// SIMATIC S7-200 project (STEP 7-Micro/WIN), CPU 224 REL 01.10

ORGANIZATION_BLOCK MAIN:OB1
TITLE=我使用这个PLC程序控制一台自动化纺织机，用于在纺织厂的织造车间。
// 系统支持多种运行模式，通过控制模式VB801选择运行模式，VB801的值必须在1到4之间。
// 程序通过高速计数器HC1记录织造的纬纱数量，计数器C10记录纬纱切换次数，用于监控生产进度和切换情况。
// 程序涉及的物理设备包括纺织机、电机、纬纱检测传感器、经纱检测传感器、启动按钮、停止按钮、纬纱切换执行器和PLC控制器。
// 系统支持多种运行模式，操作员通过控制模式选择器选择模式，其值必须在1到4之间。
// 织造通过启动按钮触发，当经纱检测传感器确认经纱正常时，运行标志置位以开始织造过程。操作员按下停止按钮时，系统复位运行标志以停止织造。纬纱切换由纬纱切换执行器控制，只有在纬纱检测传感器检测到纬纱到位时才会触发，确保切换动作准确无误。纬纱切换执行器在织造过程中由系统根据运行状态自动激活，以支持纬纱的连续切换。纬纱检测传感器用于监测纬纱的到位情况，触发计时器以协调织造节奏。系统通过经纱检测传感器监控经纱状态，若异常触发经停位标志，调用经停位子程序暂停织造。
// 为满足手动调试需求，系统支持点动控制，通过点动起输出和点动停输出实现，分别调用点动起子程序和点动停子程序，在点动模式下独立触发。若纬纱出现故障，故障标志置位，系统进入纬停状态，调用纬停位子程序安全停车并等待处理。
// 
// 
BEGIN
Network 1 // NETWORK TITLE (single line)
LD     SM0.1
CALL   初始化:SBR0
MOVB   0, MB0
?000
Network 2
LD     SM0.0
MOVB   VB93, VB153
Network 3
LDN    V142.2
MOVW   VW244, VW144
Network 4
LD     V142.2
EU
MOVW   VW144, VW244
MOVD   16#1000, VD14
R      V142.2, 1
Network 5
LDB<=  VB801, 1
=      M18.1
MOVB   1, VB801
Network 6
LDB=   VB801, 2
=      M18.2
Network 7
LDB=   VB801, 3
=      M18.3
Network 8
LDB>=  VB801, 4
=      M18.4
MOVB   4, VB801
Network 9
LD     I0.4
ED
O      M12.0
AN     T6
=      M12.0
Network 10
LD     T6
R      T6, 1
Network 11
LD     M12.0
TONR   T6, +900
Network 12
LD     I1.5
AN     M12.0
EU
CALL   启动:SBR3
Network 13
LD     I1.5
ED
CALL   即停位:SBR8
MOVD   16#20000000, VD14
Network 14
LDB=   VB811, 1
JMP    1
Network 15
LDB<>  VB811, 1
DISI
Network 16
LD     M0.0
MOVD   16#40000000, VD14
R      M0.0, 1
Network 17
// vw44 vw144 当前纬纱序号 VW244同色纬纱根数 
LD     M22.0
MOVD   16#4000000, VD14
MOVW   VW44, VW144
MOVD   &VB1000, AC3
+I     VW84, AC3
MOVB   *AC3, VB253
MOVW   +0, VW244
R      M22.0, 1
Network 18
LD     SM0.0
MOVW   VW5118, VW5116
-I     +1, VW5116
Network 19
LD     M0.1
MOVD   16#8000000, VD14
R      M0.1, 1
Network 20
LD     V228.2
MOVD   16#20000000, VD14
R      V228.2, 1
Network 21
LDB<=  VB201, 1
=      M20.1
MOVB   1, VB201
Network 22
LDB=   VB201, 2
=      M20.2
Network 23
LDB=   VB201, 3
=      M20.3
Network 24
LDB=   VB201, 4
=      M20.4
Network 25
LDB=   VB201, 5
=      M20.5
Network 26
LDB>=  VB201, 3
=      M20.3
MOVB   3, VB201
Network 27
LD     M20.1
EU
S      C10, 1
MOVW   +1, C2
MOVB   16#0, VB1101
MOVB   16#1, VB1103
Network 28
LD     M20.2
EU
S      C10, 1
S      C12, 1
MOVW   +1, C10
MOVW   +1, C12
MOVB   16#1, VB1101
MOVB   16#1, VB1103
Network 29
LD     M20.3
EU
S      C10, 1
S      C12, 1
MOVW   +2, C10
MOVW   +2, C12
MOVB   16#2, VB1101
MOVB   16#2, VB1103
Network 30
LDB=   VB231, 1
S      M18.7, 1
Network 31
LDB=   VB231, 0
R      M18.7, 1
Network 32
LD     M18.7
MOVW   VW220, VW4468
*I     +10, VW4468
Network 33
LDN    M18.7
ITD    VW220, AC0
DTR    AC0, VD1196
MOVR   VD1196, VD1192
*R     39.37, VD1192
ROUND  VD1192, VD4466
Network 34
LD     M0.2
MOVD   16#10000000, VD14
R      M0.2, 1
Network 35
LD     V160.2
MOVD   16#20000000, VD14
R      V160.2, 1
Network 36
LD     SM0.0
MOVW   VW162, VW5102
-I     +102, VW5102
MOVW   VW182, VW5108
-I     +102, VW5108
Network 37
LD     SM0.0
MOVW   VW192, VW1138
MOVW   VW192, VW1142
-I     +35, VW1142
Network 38
LD     SM0.0
MOVD   HC1, VD120
MOVD   HC1, VD5110
Network 39
LD     M0.6
MOVD   16#2000000, VD14
R      M0.6, 1
Network 40
LD     V284.2
MOVD   16#20000000, VD14
R      V284.2, 1
Network 41
LD     SM0.0
MOVW   VW286, VW1146
MOVW   VW292, VW1150
Network 42
LD     SM0.0
MOVW   VW306, VW1154
-I     +5, VW1154
MOVW   VW312, VW1158
-I     +15, VW1158
Network 43
LD     M0.3
MOVD   16#1000, VD14
R      M0.3, 1
Network 44
LD     V808.2
MOVD   16#20000000, VD14
R      V808.2, 1
Network 45
LD     M21.0
EU
R      C7, 1
MOVW   +2, C7
Network 46
LDB=   VB5115, 3
LDB=   VB201, 1
OB=    VB201, 2
ALD
=      M21.1
Network 47
LDB=   VB5115, 4
AB=    VB201, 3
=      M21.2
Network 48
LD     M21.2
EU
R      C3, 1
MOVW   +1, C3
Network 49
LDB=   VB5115, 1
OB=    VB5115, 2
AB=    VB201, 3
=      M21.4
Network 50
LD     M21.4
EU
S      C3, 1
S      C7, 1
Network 51
LDB<>  VB811, 1
END
Network 52
LBL    1
Network 53
LDN    M19.2
A      M0.3
MOVD   16#1000, VD14
R      M0.3, 1
Network 54
LD     V808.2
MOVD   16#20000000, VD14
R      V808.2, 1
Network 55
LD     SM0.0
MOVD   HC1, VD120
MOVD   HC1, VD5110
MOVW   VW122, VW864
MOVW   VW122, VW904
MOVW   VW122, VW944
MOVB   VB201, VB5115
ENI
Network 56
LD     M19.2
TON    T96, +400
Network 57
LD     I0.2
TON    T98, +5
Network 58
LDN    M10.7
A      T98
A      T96
EU
CALL   经停:SBR6
Network 59
LDN    M10.7
A      I0.1
EU
A      T96
CALL   正常停车:SBR7
Network 60
LDD>   HC1, +280
AD<    HC1, +320
S      M16.1, 1
Network 61
LDD>   HC1, +320
R      M16.1, 1
Network 62
LD     M11.5
A      M16.1
LD     I1.1
EU
LD     I0.5
EU
OLD
CTD    C11, +1
Network 63
LD     M11.2
EU
LD     C11
EU
OLD
AN     M10.7
AN     I1.5
CALL   经停位:SBR4
Network 64
LD     T98
ED
R      M11.2, 1
R      M10.6, 1
Network 65
LD     I1.1
O      I0.5
AN     M11.5
R      M11.2, 1
R      M11.4, 1
MOVD   16#20000000, VD14
Network 66
LDW>=  VW122, VW1142
AW<=   VW122, VW1138
=      M19.6
Network 67
LDN    C11
LD     M20.3
A      C13
LD     M20.2
O      M20.1
LD     M21.1
A      C13
LD     M21.3
A      C17
OLD
LDN    M21.1
AN     M21.3
OLD
ALD
OLD
ALD
ATCH   纬停:INT2, 1
ATCH   纬停:INT2, 7
LDN    I0.3
O      M11.3
ON     I0.0
ALD
S      M10.7, 1
Network 68
LDN    M19.6
DTCH   1
DTCH   7
Network 69
LD     C2
A      I0.4
TON    T97, +200
Network 70
LD     M10.7
LD     T97
EU
CTD    C10, +1
Network 71
LDD>=  HC1, +120
R      M10.5, 1
Network 72
LD     M10.7
A      M10.5
EU
AN     I1.5
CALL   纬停位:SBR5
Network 73
LD     I0.5
LPS
R      M12.6, 1
R      M11.3, 1
AN     C10
R      M10.7, 1
LRD
MOVD   16#20000000, VD14
LPP
MOVD   +0, VD1128
Network 74
LD     I0.4
ED
O      M11.1
AN     T5
=      M11.1
Network 75
LD     T5
R      T5, 1
Network 76
LD     M11.1
TONR   T5, +40
Network 77
LD     I0.5
O      M10.0
AN     M10.7
AN     M10.2
AN     M19.3
AN     M12.6
AN     M19.5
AN     T200
=      M10.0
Network 78
LDN    C10
AN     M11.5
LD     I0.5
LD     M10.0
AN     M11.1
A      I0.4
AN     I0.2
AN     I0.1
AN     M18.6
A      I1.1
OLD
ALD
AN     Q0.2
AN     Q0.3
AN     M10.2
AN     M19.3
AN     I1.4
CALL   点动起:SBR1
Network 79
LDN    I1.1
AN     I0.5
ON     T32
CALL   点动停:SBR2
Network 80
LDN    I1.1
ON     M10.0
O      M10.7
O      I0.2
O      M11.5
O      Q0.2
O      Q0.3
O      I0.1
O      M19.5
O      M19.3
O      M10.2
O      M18.6
TOF    T32, +100
Network 81
LDW>=  VW122, VW1146
AW<=   VW122, VW1150
=      M13.0
Network 82
LDN    C1
A      C10
LDN    C4
A      M11.5
OLD
A      T101
AN     M19.5
LDN    Q0.2
A      I1.3
O      Q0.3
AN     C5
OLD
AN     M13.0
AN     M10.2
AN     M19.2
AN     Q0.2
A      I0.4
=      Q0.3
Network 83
LDN    I1.4
A      C10
LD     C10
EU
LD     T38
EU
OLD
CTU    C1, +1
Network 84
LD     I1.4
EU
A      C10
A      I0.4
LD     C10
EU
CTU    C2, VW1134
Network 85
LDN    Q0.3
AN     C2
A      C10
A      C1
A      T101
TON    T38, +10
Network 86
LDN    I1.4
A      M11.5
LD     M11.5
EU
LD     T39
EU
OLD
CTU    C4, +1
Network 87
LD     I1.4
EU
A      M11.5
A      I0.4
LD     M11.5
EU
CTU    C6, VW1136
Network 88
LD     C6
A      I0.4
TON    T99, +200
Network 89
LD     T99
R      M11.5, 1
Network 90
LDN    Q0.3
AN     C6
A      M11.5
A      C4
A      T101
TON    T39, +10
Network 91
LDN    I1.4
LD     Q0.3
O      Q0.2
ALD
LDN    Q0.3
A      I1.2
LDN    Q0.2
A      I1.3
OLD
AN     M13.0
AN     M19.2
CTU    C5, +1
Network 92
LDN    Q0.3
LD     I1.2
O      Q0.2
ALD
AN     M13.0
AN     M19.2
AN     C5
A      I0.4
AN     M10.2
=      Q0.2
Network 93
LD     I1.4
A      I0.4
TON    T40, +30
Network 94
LD     Q0.2
O      Q0.3
AN     I1.4
A      I0.4
TON    T41, +30
Network 95
LD     T40
EU
LD     T41
EU
OLD
S      M10.2, 1
Network 96
LD     M11.5
ED
LPS
A      M20.3
S      M10.3, 1
LPP
LD     M20.4
O      M20.5
ALD
S      M11.6, 1
Network 97
LD     C10
ED
LD     M20.6
O      M20.5
ALD
S      M11.7, 1
Network 98
LD     M19.7
A      M10.3
LD     M10.3
EU
CTU    C3, +1
Network 99
LD     M19.7
A      M11.6
LD     M11.6
EU
CTU    C7, +2
Network 100
LD     M19.7
A      M11.7
LD     M11.7
EU
CTU    C8, +2
Network 101
LD     C7
R      M11.6, 1
Network 102
LD     C3
R      M10.3, 1
Network 103
LD     C8
R      M11.7, 1
Network 104
LD     M21.0
A      C3
EU
S      C7, 1
Network 105
LD     M21.2
A      C7
EU
S      C3, 1
Network 106
LD     M10.1
MOVB   16#AC, SMB47
MOVD   +280, SMD52
HSC    1
TON    T34, +15
TON    T36, +25
TON    T101, +15
Network 107
LDW>=  VW122, VW1154
AW<=   VW122, VW1158
=      M13.1
Network 108
LDN    I0.5
AN     I1.1
A      M10.1
TON    T200, +1800
Network 109
LD     SM0.0
MOVD   &VB1200, AC3
+I     VW244, AC3
MOVB   *AC3, VB93
Network 110
LD     SM0.0
A      C8
LD     M20.3
A      C3
LD     M20.4
A      C7
OLD
LD     M20.1
O      M20.2
LD     M21.1
A      C3
LD     M21.3
A      C7
OLD
LDN    M21.1
AN     M21.3
OLD
ALD
OLD
ALD
=      M13.2
MOVB   VB83, VB5114
DECB   VB5114
DECO   VB5114, AC1
MOVB   AC1, QB2
Network 111
LDN    M13.2
O      M10.7
O      C11
R      Q2.0, 8
Network 112
LD     SM0.0
LPS
AW=    VW244, +1
=      M13.3
LPP
AW=    VW244, VW5116
=      M13.4
Network 113
LD     Q0.2
A      I1.4
EU
O      M0.4
LPS
AN     M13.4
INCW   VW244
LRD
A      M13.4
MOVW   +1, VW244
LPP
R      M0.4, 1
Network 114
LD     Q0.3
A      I1.4
ED
O      M0.5
LPS
AN     M13.3
DECW   VW244
LRD
A      M13.3
MOVW   VW5118, VW244
-I     +1, VW244
LPP
R      M0.5, 1
Network 115
LD     M10.6
O      T98
=      Q0.5
Network 116
LD     T98
EU
LD     M10.6
EU
OLD
MOVD   16#400, VD14
Network 117
LD     M10.7
EU
MOVD   16#200, VD14
Network 118
LD     M10.7
LD     M18.6
A      SM0.5
OLD
=      Q0.6
Network 119
LD     M11.4
EU
MOVD   16#800, VD14
Network 120
LD     M11.4
=      Q0.7
Network 121
LD     M19.5
O      M19.3
O      M10.2
O      M12.6
=      Q1.0
Network 122
LD     M10.2
EU
MOVD   16#10000, VD14
Network 123
LD     M19.3
MOVD   16#80, VD14
Network 124
LD     M19.5
MOVD   16#20, VD14
Network 125
LD     M10.5
AN     SM0.4
LD     SM0.4
ED
CTU    C15, +500
Network 126
LD     SM0.4
EU
MOVW   C15, VW132
*I     +2, VW132
Network 127
LD     M19.2
AN     M10.5
AN     I1.5
TON    T35, +200
Network 128
LD     M19.2
A      M10.5
AN     I1.5
TON    T33, +200
Network 129
LD     T35
O      T33
S      M19.3, 1
Network 130
LD     M19.3
EU
CALL   即停位:SBR8
Network 131
LD     T34
EU
MOVD   HC1, VD1116
Network 132
LD     T36
EU
MOVD   HC1, VD1128
-D     VD1116, VD1128
Network 133
LD     M10.1
AD>=   VD1128, +5
=      M19.5
Network 134
LD     M10.7
LPS
R      M11.5, 1
S      C4, 1
S      C6, 1
R      M11.2, 1
A      M20.3
S      C3, 1
LPP
LD     M20.4
O      M20.5
ALD
S      C7, 1
Network 135
LD     M19.2
AN     I0.4
EU
CALL   经停位:SBR4
S      M12.6, 1
Network 136
LD     M19.2
A      M18.6
EU
CALL   经停位:SBR4
Network 137
LD     M12.6
EU
S      C3, 1
R      C10, 1
S      C7, 2
Network 138
LD     C127
LDB=   VB1053, 0
CTU    C128, +32765
Network 139
LD     M10.5
LDB=   VB1053, 0
LD     C127
EU
OLD
CTU    C127, +32767
Network 140
LD     C129
LDB=   VB1073, 0
CTU    C130, +32765
Network 141
LD     M10.5
LDB=   VB1073, 0
LD     C129
EU
OLD
CTU    C129, +32767
Network 142
LDW>=  VW1064, VW210
=      M18.6
END_ORGANIZATION_BLOCK

SUBROUTINE_BLOCK 初始化:SBR0
TITLE= 
// SUBROUTINE COMMENTS
// Press F1 for help and example program
//  
BEGIN
Network 1 // NETWORK TITLE (single line)
//  
// NETWORK COMMENTS
//  
// 
LD     SM0.0
MOVB   16#EC, SMB47
HDEF   1, 10
MOVD   VD5110, SMD48
MOVD   +280, SMD52
HSC    1
END_SUBROUTINE_BLOCK

SUBROUTINE_BLOCK 点动起:SBR1
TITLE=
BEGIN
Network 1
LD     SM0.0
MOVB   16#DB, SMB67
MOVW   +200, SMW68
MOVW   +100, SMW70
PLS    0
MOVW   16#DA, SMW67
END_SUBROUTINE_BLOCK

SUBROUTINE_BLOCK 点动停:SBR2
TITLE=
BEGIN
Network 1
LD     SM0.0
MOVW   +0, SMW70
PLS    0
MOVW   16#DA, SMW67
END_SUBROUTINE_BLOCK

SUBROUTINE_BLOCK 启动:SBR3
TITLE=
BEGIN
Network 1
LD     SM0.0
MOVB   16#DB, SMB77
MOVW   +30000, SMW78
MOVW   +30000, SMW80
PLS    1
MOVW   16#DA, SMW77
Network 2
LD     SM0.0
S      M19.2, 1
R      M10.1, 1
END_SUBROUTINE_BLOCK

SUBROUTINE_BLOCK 经停位:SBR4
TITLE=
BEGIN
Network 1
LD     SM0.0
MOVB   16#AC, SMB47
MOVD   VD5106, SMD52
HSC    1
ATCH   停车:INT0, 13
END_SUBROUTINE_BLOCK

SUBROUTINE_BLOCK 纬停位:SBR5
TITLE=
BEGIN
Network 1
LD     SM0.0
MOVB   16#AC, SMB47
MOVD   VD5100, SMD52
HSC    1
ATCH   停车:INT0, 13
END_SUBROUTINE_BLOCK

SUBROUTINE_BLOCK 经停:SBR6
TITLE=
BEGIN
Network 1
LD     M20.2
O      M20.3
O      M20.4
O      M20.5
S      M11.5, 1
Network 2
LD     M20.1
O      M20.6
S      M11.2, 1
Network 3
LD     SM0.0
S      M10.6, 1
END_SUBROUTINE_BLOCK

SUBROUTINE_BLOCK 正常停车:SBR7
TITLE=
BEGIN
Network 1
LD     M20.1
O      M20.6
S      M11.2, 1
Network 2
LD     M20.2
O      M20.3
O      M20.4
O      M20.5
S      M11.5, 1
Network 3
LD     SM0.0
S      M11.4, 1
END_SUBROUTINE_BLOCK

SUBROUTINE_BLOCK 即停位:SBR8
TITLE=
BEGIN
Network 1
LD     SM0.0
MOVW   +0, SMW80
PLS    1
MOVW   16#DA, SMW77
S      M10.1, 1
R      M19.2, 1
END_SUBROUTINE_BLOCK

INTERRUPT_BLOCK 停车:INT0
TITLE= 
// INTERRUPT ROUTINE COMMENTS
// Press F1 for help and example program
//  
BEGIN
Network 1 // NETWORK TITLE (single line)
//  
// NETWORK COMMENTS
//  
// 
LD     SM0.0
MOVW   +0, SMW80
PLS    1
MOVW   16#DA, SMW77
S      M10.1, 1
R      M19.2, 1
Network 2
LD     SM0.0
CRETI
END_INTERRUPT_BLOCK

INTERRUPT_BLOCK 纬停:INT2
TITLE=
BEGIN
Network 1
LD     SM0.0
S      M11.3, 1
S      M10.7, 1
Network 2
LD     SM0.0
CRETI
END_INTERRUPT_BLOCK

DATA_BLOCK_TAB USER1
BEGIN
//BEGIN TD200_BLOCK 0
// 
//(Comments within this block should not be edited or removed)
// 
VB0      'TD'
VB2      16#60               //Set Language to Chinese, set Update to as fast as possible 
VB3      16#E1               //Set the display to 40 character mode; Up key V3.2; Down key V3.3;
VB4      27                  //Set the number of messages
VB5      0                   //Set the Function Keys notification bits to M0.0 - M0.7
VW6      34                  //Set the starting address for messages to  VW34
VW8      14                  //Set the starting address for message enable bits to VW14
VW10     1234                //Global Password (if enabled)
VW12     256                 //Character Set = Simplified Chinese
//MESSAGE 1
//Message Enable Bit V14.7 
VB34     '      杭    州      方大电子技术开发公司'
//MESSAGE 2
//Message Enable Bit V14.6 
VB74     '选色序号'
VB82     16#10               //Edit Notification V82.2; No Acknowledgement;No Password;
VB83     16#10               //Signed Word; 0 Digits to the right of the decimal;
VW84     16#0                //Embedded Data Value: Move data for display here.
VB86     '色号'
VB90     16#0                //No Edit;No Acknowledgement;No Password;
VB91     16#10               //Signed Word; 0 Digits to the right of the decimal;
VW92     16#0                //Embedded Data Value: Move data for display here.
VB94     '同色纬数'
VB102    16#0                //No Edit;No Acknowledgement;No Password;
VB103    16#10               //Signed Word; 0 Digits to the right of the decimal;
VW104    16#0                //Embedded Data Value: Move data for display here.
VB106    '        '
//MESSAGE 3
//Message Enable Bit V14.5 
VB114    '角度'
VB118    16#0                //No Edit;No Acknowledgement;No Password;
VB119    16#20               //Signed Double Word; 0 Digits to the right of the decimal;
VD120    16#0                //Embedded Data Value: Move data for display here.
VB124    '  速度'
VB130    16#0                //No Edit;No Acknowledgement;No Password;
VB131    16#10               //Signed Word; 0 Digits to the right of the decimal;
VW132    16#0                //Embedded Data Value: Move data for display here.
VB134    '当前序号'
VB142    16#10               //Edit Notification V142.2; No Acknowledgement;No Password;
VB143    16#10               //Signed Word; 0 Digits to the right of the decimal;
VW144    16#0                //Embedded Data Value: Move data for display here.
VB146    '色号'
VB150    16#0                //No Edit;No Acknowledgement;No Password;
VB151    16#10               //Signed Word; 0 Digits to the right of the decimal;
VW152    16#0                //Embedded Data Value: Move data for display here.
//MESSAGE 4
//Message Enable Bit V14.4 
VB154    '纬停角'
VB160    16#10               //Edit Notification V160.2; No Acknowledgement;No Password;
VB161    16#10               //Signed Word; 0 Digits to the right of the decimal;
VW162    16#0                //Embedded Data Value: Move data for display here.
VB164    '    探纬角经停角'
VB180    16#10               //Edit Notification V180.2; No Acknowledgement;No Password;
VB181    16#10               //Signed Word; 0 Digits to the right of the decimal;
VW182    16#0                //Embedded Data Value: Move data for display here.
VB184    '      '
VB190    16#10               //Edit Notification V190.2; No Acknowledgement;No Password;
VB191    16#10               //Signed Word; 0 Digits to the right of the decimal;
VW192    16#0                //Embedded Data Value: Move data for display here.
//MESSAGE 5
//Message Enable Bit V14.3 
VB194    '程式'
VB198    16#10               //Edit Notification V198.2; No Acknowledgement;No Password;
VB199    16#10               //Signed Word; 0 Digits to the right of the decimal;
VW200    16#0                //Embedded Data Value: Move data for display here.
VB202    '  落布'
VB208    16#10               //Edit Notification V208.2; No Acknowledgement;No Password;
VB209    16#10               //Signed Word; 0 Digits to the right of the decimal;
VW210    16#0                //Embedded Data Value: Move data for display here.
VB212    '  纬密'
VB218    16#10               //Edit Notification V218.2; No Acknowledgement;No Password;
VB219    16#10               //Signed Word; 0 Digits to the right of the decimal;
VW220    16#0                //Embedded Data Value: Move data for display here.
VB222    '  单位'
VB228    16#10               //Edit Notification V228.2; No Acknowledgement;No Password;
VB229    16#10               //Signed Word; 0 Digits to the right of the decimal;
VW230    16#0                //Embedded Data Value: Move data for display here.
VB232    '  '
//MESSAGE 6
//Message Enable Bit V14.2 
VB234    '选色序号'
VB242    16#0                //No Edit;No Acknowledgement;No Password;
VB243    16#10               //Signed Word; 0 Digits to the right of the decimal;
VW244    16#0                //Embedded Data Value: Move data for display here.
VB246    '色号'
VB250    16#10               //Edit Notification V250.2; No Acknowledgement;No Password;
VB251    16#10               //Signed Word; 0 Digits to the right of the decimal;
VW252    16#0                //Embedded Data Value: Move data for display here.
VB254    '同色纬数'
VB262    16#10               //Edit Notification V262.2; No Acknowledgement;No Password;
VB263    16#10               //Signed Word; 0 Digits to the right of the decimal;
VW264    16#0                //Embedded Data Value: Move data for display here.
VB266    '        '
//MESSAGE 7
//Message Enable Bit V14.1 
VB274    '禁止倒综区'
VB284    16#10               //Edit Notification V284.2; No Acknowledgement;No Password;
VB285    16#10               //Signed Word; 0 Digits to the right of the decimal;
VW286    16#0                //Embedded Data Value: Move data for display here.
VB288    '到'
VB290    16#10               //Edit Notification V290.2; No Acknowledgement;No Password;
VB291    16#10               //Signed Word; 0 Digits to the right of the decimal;
VW292    16#0                //Embedded Data Value: Move data for display here.
VB294    '选色保护区'
VB304    16#10               //Edit Notification V304.2; No Acknowledgement;No Password;
VB305    16#10               //Signed Word; 0 Digits to the right of the decimal;
VW306    16#0                //Embedded Data Value: Move data for display here.
VB308    '到'
VB310    16#10               //Edit Notification V310.2; No Acknowledgement;No Password;
VB311    16#10               //Signed Word; 0 Digits to the right of the decimal;
VW312    16#0                //Embedded Data Value: Move data for display here.
//MESSAGE 8
//Message Enable Bit V14.0 
VB314    '甲班产量'
VB322    16#0                //No Edit;No Acknowledgement;No Password;
VB323    16#10               //Signed Word; 0 Digits to the right of the decimal;
VW324    16#0                //Embedded Data Value: Move data for display here.
VB326    '  米    断经'
VB338    16#0                //No Edit;No Acknowledgement;No Password;
VB339    16#10               //Signed Word; 0 Digits to the right of the decimal;
VW340    16#0                //Embedded Data Value: Move data for display here.
VB342    '    断纬'
VB350    16#0                //No Edit;No Acknowledgement;No Password;
VB351    16#10               //Signed Word; 0 Digits to the right of the decimal;
VW352    16#0                //Embedded Data Value: Move data for display here.
//MESSAGE 9
//Message Enable Bit V15.7 
VB354    '乙班产量'
VB362    16#0                //No Edit;No Acknowledgement;No Password;
VB363    16#10               //Signed Word; 0 Digits to the right of the decimal;
VW364    16#0                //Embedded Data Value: Move data for display here.
VB366    '  米    断经'
VB378    16#0                //No Edit;No Acknowledgement;No Password;
VB379    16#10               //Signed Word; 0 Digits to the right of the decimal;
VW380    16#0                //Embedded Data Value: Move data for display here.
VB382    '    断纬'
VB390    16#0                //No Edit;No Acknowledgement;No Password;
VB391    16#10               //Signed Word; 0 Digits to the right of the decimal;
VW392    16#0                //Embedded Data Value: Move data for display here.
//MESSAGE 10
//Message Enable Bit V15.6 
VB394    '丙班产量'
VB402    16#0                //No Edit;No Acknowledgement;No Password;
VB403    16#10               //Signed Word; 0 Digits to the right of the decimal;
VW404    16#0                //Embedded Data Value: Move data for display here.
VB406    '  米    断经'
VB418    16#0                //No Edit;No Acknowledgement;No Password;
VB419    16#10               //Signed Word; 0 Digits to the right of the decimal;
VW420    16#0                //Embedded Data Value: Move data for display here.
VB422    '    断纬'
VB430    16#0                //No Edit;No Acknowledgement;No Password;
VB431    16#10               //Signed Word; 0 Digits to the right of the decimal;
VW432    16#0                //Embedded Data Value: Move data for display here.
//MESSAGE 11
//Message Enable Bit V15.5 
VB434    '丁班产量'
VB442    16#0                //No Edit;No Acknowledgement;No Password;
VB443    16#10               //Signed Word; 0 Digits to the right of the decimal;
VW444    16#0                //Embedded Data Value: Move data for display here.
VB446    '  米    断经'
VB458    16#0                //No Edit;No Acknowledgement;No Password;
VB459    16#10               //Signed Word; 0 Digits to the right of the decimal;
VW460    16#0                //Embedded Data Value: Move data for display here.
VB462    '    断纬'
VB470    16#0                //No Edit;No Acknowledgement;No Password;
VB471    16#10               //Signed Word; 0 Digits to the right of the decimal;
VW472    16#0                //Embedded Data Value: Move data for display here.
//MESSAGE 12
//Message Enable Bit V15.4 
VB474    '启动信号OK！                            '
//MESSAGE 13
//Message Enable Bit V15.3 
VB514    '停止信号OK！                            '
//MESSAGE 14
//Message Enable Bit V15.2 
VB554    '前寻纬信号OK！                          '
//MESSAGE 15
//Message Enable Bit V15.1 
VB594    '后纬寻信号OK！                          '
//MESSAGE 16
//Message Enable Bit V15.0 
VB634    '多臂机触点故障！                        '
//MESSAGE 17
//Message Enable Bit V16.7 
VB674    '断经信号OK！                            '
//MESSAGE 18
//Message Enable Bit V16.6 
VB714    '断纬信号OK！                            '
//MESSAGE 19
//Message Enable Bit V16.5 
VB754    '重纬信号OK！                            '
//MESSAGE 20
//Message Enable Bit V16.4 
VB794    '班次'
VB798    16#10               //Edit Notification V798.2; No Acknowledgement;No Password;
VB799    16#10               //Signed Word; 0 Digits to the right of the decimal;
VW800    16#0                //Embedded Data Value: Move data for display here.
VB802    '  状态'
VB808    16#10               //Edit Notification V808.2; No Acknowledgement;No Password;
VB809    16#10               //Signed Word; 0 Digits to the right of the decimal;
VW810    16#0                //Embedded Data Value: Move data for display here.
VB812    '                      '
//MESSAGE 21
//Message Enable Bit V16.3 
VB834    '正常停车!           当前角度'
VB862    16#0                //No Edit;No Acknowledgement;No Password;
VB863    16#10               //Signed Word; 0 Digits to the right of the decimal;
VW864    16#0                //Embedded Data Value: Move data for display here.
VB866    '        '
//MESSAGE 22
//Message Enable Bit V16.2 
VB874    '断经停车!           当前角度'
VB902    16#0                //No Edit;No Acknowledgement;No Password;
VB903    16#10               //Signed Word; 0 Digits to the right of the decimal;
VW904    16#0                //Embedded Data Value: Move data for display here.
VB906    '        '
//MESSAGE 23
//Message Enable Bit V16.1 
VB914    '断纬或重纬停车 !    当前角度'
VB942    16#0                //No Edit;No Acknowledgement;No Password;
VB943    16#10               //Signed Word; 0 Digits to the right of the decimal;
VW944    16#0                //Embedded Data Value: Move data for display here.
VB946    '        '
//MESSAGE 24
//Message Enable Bit V16.0 
VB954    '点动信号OK!                             '
//MESSAGE 25
//Message Enable Bit V17.7 
VB994    '离合器故障！                            '
//MESSAGE 26
//Message Enable Bit V17.6 
VB1034   '总产量  '
VB1042   16#0                //No Edit;No Acknowledgement;No Password;
VB1043   16#10               //Signed Word; 0 Digits to the right of the decimal;
VW1044   16#0                //Embedded Data Value: Move data for display here.
VB1046   '清零'
VB1050   16#10               //Edit Notification V1050.2; No Acknowledgement;No Password;
VB1051   16#10               //Signed Word; 0 Digits to the right of the decimal;
VW1052   16#0                //Embedded Data Value: Move data for display here.
VB1054   '布长    '
VB1062   16#0                //No Edit;No Acknowledgement;No Password;
VB1063   16#10               //Signed Word; 0 Digits to the right of the decimal;
VW1064   16#0                //Embedded Data Value: Move data for display here.
VB1066   '清零'
VB1070   16#10               //Edit Notification V1070.2; No Acknowledgement;No Password;
VB1071   16#10               //Signed Word; 0 Digits to the right of the decimal;
VW1072   16#0                //Embedded Data Value: Move data for display here.
//MESSAGE 27
//Message Enable Bit V17.5 
VB1074   '刹车不灵敏！                            '
//END TD200_BLOCK 0
END_DATA_BLOCK_TAB
